(* Logix 5000 project; controller cal1615 1756-L62 rev 20.11; software revision 20.05 *)

TASK MainTask (continuous, watchdog 500 ms) : P01_System, P02_MOP_HMI_Iface, P11_Zone_1, P12_Zone_2, P13_Zone_3, P19_Advanced_Cooling, P20_Letoff, P21_Splice_Press, P22_Tension_Stand_1
TASK PIDE (periodic, rate 100 ms, priority 10, watchdog 500 ms) : P01_Main

MODULES
   Local : 1756-L62 (ICP 0, rev 20.11)
      p00_di_01 : 1756-IB16 (ICP 4, rev 3.1, Input RPI 20 ms)
           Local:4:I.DATA.0   // Digital Input Zone 1 Burner Auto
           Local:4:I.DATA.1   // Digital Input Zone 1 High Temperature Limit is Ok
           Local:4:I.DATA.2   // Digital Input Zone 1 Burner Safeties Ok
           Local:4:I.DATA.3   // Digital Input Zone 1 Recirculation Fan Rotating
           Local:4:I.DATA.4   // Digital Input Zone 1 Exhaust Fan Rotating
           Local:4:I.DATA.5   // Digital Input Zone 1 Flame Failure
           Local:4:I.DATA.6   // Digital Input Zone 1 Burner is On
           Local:4:I.DATA.7   // Digital Input Zone 1 Spare
           Local:4:I.DATA.8   // Digital Input Zone 2 Burner Auto
           Local:4:I.DATA.9   // Digital Input Zone 2 High Temperature Limit is Ok
           Local:4:I.DATA.10   // Digital Input Zone 2 Burner Safeties Ok
           Local:4:I.DATA.11   // Digital Input Zone 2 Recirculation Fan Rotating
           Local:4:I.DATA.12   // Digital Input Zone 2 Exhaust Fan Rotating
           Local:4:I.DATA.13   // Digital Input Zone 2 Flame Failure
           Local:4:I.DATA.14   // Digital Input Zone 2 Burner is On
           Local:4:I.DATA.15   // Digital Input Zone 2 Spare
      p00_di_02 : 1756-IB16 (ICP 5, rev 3.1, Input RPI 20 ms)
           Local:5:I.DATA.0   // Digital Input Zone 3 Recirculation Fan Rotating
           Local:5:I.DATA.1   // Digital Input Zone 3 Exhaust Fan Rotating
           Local:5:I.DATA.2   // Digital Input Zone 3 Spare
           Local:5:I.DATA.3   // Digital Input Zone 3 Spare
           Local:5:I.DATA.4   // Digital Input Zone 3 Spare
           Local:5:I.DATA.5   // Digital Input Zone 3 Spare
           Local:5:I.DATA.6   // Digital Input Zone 3 Spare
           Local:5:I.DATA.7   // Digital Input Zone 3 Spare
           Local:5:I.DATA.8   // Digital Input Rope Switch 1 Active
           Local:5:I.DATA.9   // Digital Input Rope Switch 2 Active
           Local:5:I.DATA.10   // Digital Input Rope Switch 3 Active
           Local:5:I.DATA.11   // Digital Input Rope Switch 4 Active
           Local:5:I.DATA.12   // Digital Input Rope Switch 5 Active
           Local:5:I.DATA.13   // Digital Input Rope Switch 6 Active
           Local:5:I.DATA.14   // Digital Input Rope Switch 7 Active
           Local:5:I.DATA.15   // Digital Input Rope Switch 8 Active
      p00_di_03 : 1756-IB16 (ICP 6, rev 3.1, Input RPI 20 ms)
           Local:6:I.DATA.0   // Digital Input Main HMI Reset PB
           Local:6:I.DATA.1   // Digital Input Main HMI Estop PB
           Local:6:I.DATA.2   // Digital Input Safety Relay 1 OK
           Local:6:I.DATA.3   // Digital Input Safety Relay 2 OK
           Local:6:I.DATA.4   // Digital Input Two Hand Safety Relay
           Local:6:I.DATA.5   // Digital Input Splice Plate High Temperature
           Local:6:I.DATA.6   // Digital Input Spare
           Local:6:I.DATA.7   // Digital Input Retraction and Rotation Fault
           Local:6:I.DATA.8   // Digital Input Spare
           Local:6:I.DATA.9   // Digital Input Spare
           Local:6:I.DATA.10   // Digital Input Spare
           Local:6:I.DATA.11   // Digital Input Spare
           Local:6:I.DATA.12   // Digital Input Spare
           Local:6:I.DATA.13   // Digital Input Spare
           Local:6:I.DATA.14   // Digital Input Spare
           Local:6:I.DATA.15   // Digital Input Spare
      p00_do_01 : 1756-OA16I (ICP 7, rev 3.1, Output RPI 20 ms)
           Local:7:O.DATA.0   // Digital Output Zone 1 Burner Enable
           Local:7:O.DATA.1   // Digital Output Zone 1 Burner Reset
           Local:7:O.DATA.2   // Digital Output Zone 2 Burner Enable
           Local:7:O.DATA.3   // Digital Output Zone 2 Burner Reset
           Local:7:O.DATA.4   // Digital Output Retraction System Motion
           Local:7:O.DATA.5   // Digital Output Spare
           Local:7:O.DATA.6   // Digital Output Spare
           Local:7:O.DATA.7   // Digital Output Spare
           Local:7:O.DATA.8   // Digital Output Spare
           Local:7:O.DATA.9   // Digital Output Spare
           Local:7:O.DATA.10   // Digital Output Spare
           Local:7:O.DATA.11   // Digital Output Spare
           Local:7:O.DATA.12   // Digital Output Spare
           Local:7:O.DATA.13   // Digital Output Spare
           Local:7:O.DATA.14   // Digital Output Spare
           Local:7:O.DATA.15   // Digital Output Spare
      Enet_A : 1756-ENBT (Ethernet 10.0.0.1, ICP 1, rev 4.1)
         p00_io_letoff : 1794-AENT (Ethernet 10.0.0.10, rev 3.1, Output RPI 25 ms)
            p00_io_letoff_di_04 : 1794-IB16 (Flex 7, rev 1.1)
                 p00_io_letoff:7:I.0   // Digital Input Impreg PB: Splice Jump
                 p00_io_letoff:7:I.1   // Digital Input Impreg SSS: Metering Rolls Open
                 p00_io_letoff:7:I.2   // Digital Input Impreg SSS: Metering Rolls Close
                 p00_io_letoff:7:I.3   // Digital Input Impreg SSS: Metering Rolls Jog FWD
                 p00_io_letoff:7:I.4   // Digital Input Impreg SSS: Metering Rolls Jog REV
                 p00_io_letoff:7:I.5   // Digital Input Impreg PP: EStop Active
                 p00_io_letoff:7:I.6   // Digital Input Impreg Spare
                 p00_io_letoff:7:I.7   // Digital Input Impreg Spare
                 p00_io_letoff:7:I.8   // Digital Input Impreg PR: Dip Tank Up
                 p00_io_letoff:7:I.9   // Digital Input Impreg PS: Enclosure Supply Filter Dirty
                 p00_io_letoff:7:I.10   // Digital Input Impreg Enclosure Supply Fan Rotating
                 p00_io_letoff:7:I.11   // Digital Input Impreg Through Tank Level Low
                 p00_io_letoff:7:I.12   // Digital Input Impreg Tank Level High
                 p00_io_letoff:7:I.13   // Digital Input Impreg Tank Level Low
                 p00_io_letoff:7:I.14   // Digital Input Impreg Spare
                 p00_io_letoff:7:I.15   // Digital Input Impreg Spare
            p00_io_letoff_do_01 : vendor 1 type 7 code 35 (Flex 3, rev 1.1)
                 p00_io_letoff:3:O.0   // Digital Output Letoff B Selected
                 p00_io_letoff:3:O.1   // Digital Output Letoff A Selected
                 p00_io_letoff:3:O.2   // Digital Output Letoff Turret in position
                 p00_io_letoff:3:O.3   // Digital Output Letoff Spare
                 p00_io_letoff:3:O.4   // Digital Output Splice Press Inlet Clamp Close
                 p00_io_letoff:3:O.5   // Digital Output Splice Press Platen Close
                 p00_io_letoff:3:O.7   // Digital Output Splice Press Exit Clamp Close
                 p00_io_letoff:3:O.8   // Digital Output Letoff Accumulator Feedroll Clutch On
                 p00_io_letoff:3:O.9   // Digital Output Letoff Accumulator Feedroll Nip Close
                 p00_io_letoff:3:O.10   // Digital Output Letoff Accumulator Tension On
                 p00_io_letoff:3:O.11   // Digital Output Letoff Accumulator Tension High/Low
                 p00_io_letoff:3:O.12   // Digital Output Tension Stand 1 Nip Close
                 p00_io_letoff:3:O.13   // Digital Output Spare
                 p00_io_letoff:3:O.14   // Digital Output Impreg Metering Rolls Close
                 p00_io_letoff:3:O.15   // Digital Output Spare
            p00_io_letoff_di_01 : 1794-IB16 (Flex 4, rev 1.1)
                 p00_io_letoff:4:I.0   // Digital Input Letoff SS: Letoff A Selected
                 p00_io_letoff:4:I.1   // Digital Input Letoff PB: Letoff A On
                 p00_io_letoff:4:I.2   // Digital Input Letoff PB: Letoff A Off Off=0
                 p00_io_letoff:4:I.3   // Digital Input Letoff PB: Letoff A Jog FWD
                 p00_io_letoff:4:I.4   // Digital Input Letoff PB: Letoff A Jog REV
                 p00_io_letoff:4:I.5   // Digital Input Letoff PB: Letoff B On
                 p00_io_letoff:4:I.6   // Digital Input Letoff PB: Letoff B Off
                 p00_io_letoff:4:I.7   // Digital Input Letoff PB: Letoff B Jog FWD
                 p00_io_letoff:4:I.8   // Digital Input Letoff PB: Letoff B Jog REV
                 p00_io_letoff:4:I.9   // Digital Input Letoff PB: Turret FWD
                 p00_io_letoff:4:I.10   // Digital Input Letoff PB: Turret REV
                 p00_io_letoff:4:I.11   // Digital Input Letoff PP: Estop Active
                 p00_io_letoff:4:I.12   // Digital Input Letoff Spare
                 p00_io_letoff:4:I.13   // Digital Input Letoff Turret in Position
                 p00_io_letoff:4:I.14   // Digital Input Letoff Spare
                 p00_io_letoff:4:I.15   // Digital Input Letoff Spare
            p00_io_letoff_di_02 : 1794-IB16 (Flex 5, rev 1.1)
                 p00_io_letoff:5:I.0   // Digital Input Splice Press Spare
                 p00_io_letoff:5:I.1   // Digital Input Splice Press Spare
                 p00_io_letoff:5:I.2   // Digital Input Splice Press PB: Open Platen
                 p00_io_letoff:5:I.3   // Digital Input Splice Press PB: Close Inlet Clamp
                 p00_io_letoff:5:I.4   // Digital Input Splice Press PB: Close Exit Clamp
                 p00_io_letoff:5:I.5   // Digital Input Splice Press PB: Feedroll Jog FWD
                 p00_io_letoff:5:I.6   // Digital Input Splice Press PB: Feedroll Jog REV
                 p00_io_letoff:5:I.7   // Digital Input Splice Press PB: Close Feedroll Nip
                 p00_io_letoff:5:I.8   // Digital Input Splice Press PB: Fill Letoff Accumulator
                 p00_io_letoff:5:I.9   // Digital Input Splice Press PP: EStop Active
                 p00_io_letoff:5:I.10   // Digital Input Splice Press Spare
                 p00_io_letoff:5:I.11   // Digital Input Accumulator Door Open
                 p00_io_letoff:5:I.12   // Digital Input Splice Press Spare
                 p00_io_letoff:5:I.13   // Digital Input Splice Press Spare
                 p00_io_letoff:5:I.14   // Digital Input Splice Press LS: Platen Closed
                 p00_io_letoff:5:I.15   // Digital Input Splice Press Spare
            p00_io_letoff_di_03 : 1794-IB16 (Flex 6, rev 1.1)
                 p00_io_letoff:6:I.0   // Digital Input Letoff Accumulator LS: Upper Limit Active
                 p00_io_letoff:6:I.1   // Digital Input Letoff Accumulator LS: Lower Limit Active
                 p00_io_letoff:6:I.2   // Digital Input Letoff Accumulator Spare
                 p00_io_letoff:6:I.3   // Digital Input Letoff Accumulator PB: Tension Stand 1 Jog FWD
                 p00_io_letoff:6:I.4   // Digital Input Letoff Accumulator PB: Tension Stand 1 Jog REV
                 p00_io_letoff:6:I.5   // Digital Input Letoff Accumulator SS: Tension Stand 1 Jog/Thread/Run Jog
                 p00_io_letoff:6:I.6   // Digital Input Letoff Accumulator SS: Tension Stand 1 Jog/Thread/Run Run
                 p00_io_letoff:6:I.7   // Digital Input Letoff Accumulator SS: Tension Stand 1 Nip Open/Auto/Close Open
                 p00_io_letoff:6:I.8   // Digital Input Letoff Accumulator SS: Tension Stand 1 Nip Open/Auto/Close Close
                 p00_io_letoff:6:I.9   // Digital Input Letoff Accumulator PP: EStop Active
                 p00_io_letoff:6:I.10   // Digital Input Letoff Accumulator Spare
                 p00_io_letoff:6:I.11   // Digital Input Letoff Accumulator Spare
                 p00_io_letoff:6:I.12   // Digital Input Letoff Accumulator Spare
                 p00_io_letoff:6:I.13   // Digital Input Letoff Accumulator Spare
                 p00_io_letoff:6:I.14   // Digital Input Letoff Accumulator Spare
                 p00_io_letoff:6:I.15   // Digital Input Letoff Accumulator Spare
            p00_io_letoff_ao_01 : 1794-OE4 (Flex 0, rev 2.1, Output RPI 80 ms)
                 p00_io_letoff:0:O.CH0DATA   // Analog Output Letoff Accumulator Counter Pressure
                 p00_io_letoff:0:O.CH1DATA   // Analog Output Letoff Accumulator Tension Pressure
                 p00_io_letoff:0:O.CH2DATA   // Analog Output Letoff Accumulator Fill Pressure
                 p00_io_letoff:0:O.CH3DATA   // Analog Output Letoff Spare
            p00_io_letoff_ai_01 : vendor 1 type 10 code 25 (Flex 1, rev 2.1, Input RPI 80 ms)
                 p00_io_letoff:1:I.CH0DATA   // Analog Input Letoff Roll Diameter
                 p00_io_letoff:1:I.CH1DATA   // Analog Input Letoff Accumulator Position
                 p00_io_letoff:1:I.CH2DATA   // Analog Input Impreg Enclosure LEL Level
                 p00_io_letoff:1:I.CH3DATA   // Analog Input Impreg Enclosure Static Pressure
                 p00_io_letoff:1:I.CH4DATA   // Analog Input Impreg Enclosure to Zone 1 Differential Pressure
                 p00_io_letoff:1:I.CH5DATA   // Analog Input Spare
                 p00_io_letoff:1:I.CH6DATA   // Analog Input Spare
                 p00_io_letoff:1:I.CH7DATA   // Analog Input Spare
            p00_io_letoff_tc_01 : vendor 1 type 10 code 28 (Flex 2, rev 1.1, Input RPI 80 ms)
                 p00_io_letoff:2:I.CH0DATA   // Thermocouple Input Splicer Platen Temperature
                 p00_io_letoff:2:I.CH1DATA   // Thermocouple Input Spare
                 p00_io_letoff:2:I.CH2DATA   // Thermocouple Input Spare
                 p00_io_letoff:2:I.CH3DATA   // Thermocouple Input Spare
                 p00_io_letoff:2:I.CH4DATA   // Thermocouple Input Spare
                 p00_io_letoff:2:I.CH5DATA   // Thermocouple Input Spare
                 p00_io_letoff:2:I.CH6DATA   // Thermocouple Input Spare
                 p00_io_letoff:2:I.CH7DATA   // Thermocouple Input Spare
                 p00_io_letoff:2:I.CH0OVERRANGEALARM   // Analog Input Splice Press TC Open Wire
                 p00_io_letoff:2:I.CH1OVERRANGEALARM   // Analog Input Spare TC Open Wire
                 p00_io_letoff:2:I.CH2OVERRANGEALARM   // Analog Input Spare TC Open Wire
                 p00_io_letoff:2:I.CH3OVERRANGEALARM   // Analog Input Spare TC Open Wire
                 p00_io_letoff:2:I.CH4OVERRANGEALARM   // Analog Input Spare TC Open Wire
                 p00_io_letoff:2:I.CH5OVERRANGEALARM   // Analog Input Spare TC Open Wire
                 p00_io_letoff:2:I.CH6OVERRANGEALARM   // Analog Input Spare TC Open Wire
                 p00_io_letoff:2:I.CH7OVERRANGEALARM   // Analog Input Spare TC Open Wire
         p00_io_oven : 1794-AENT (Ethernet 10.0.0.11, rev 3.1, Output RPI 25 ms)
            p00_io_oven_di_03 : 1794-IB16 (Flex 5, rev 1.1)
                 p00_io_oven:5:I.0   // Digital Input LS: Safety Pin 1 Stowed
                 p00_io_oven:5:I.1   // Digital Input LS: Safety Pin 2 Stowed
                 p00_io_oven:5:I.2   // Digital Input LS: Safety Pin 3 Stowed
                 p00_io_oven:5:I.3   // Digital Input LS: Safety Pin 4 Stowed
                 p00_io_oven:5:I.4   // Digital Input LS: Safety Pin 5 Stowed
                 p00_io_oven:5:I.5   // Digital Input LS: Safety Pin 6 Stowed
                 p00_io_oven:5:I.6   // Digital Input LS: Safety Pin 7 Stowed
                 p00_io_oven:5:I.7   // Digital Input LS: Safety Pin 8 Stowed
                 p00_io_oven:5:I.8   // Digital Input Spare
                 p00_io_oven:5:I.9   // Digital Input Spare
                 p00_io_oven:5:I.10   // Digital Input Spare
                 p00_io_oven:5:I.11   // Digital Input Spare
                 p00_io_oven:5:I.12   // Digital Input Spare
                 p00_io_oven:5:I.13   // Digital Input Spare
                 p00_io_oven:5:I.14   // Digital Input Spare
                 p00_io_oven:5:I.15   // Digital Input Spare
                 p00_io_oven:5:I   // Digital Input Safety Pins Stowed
            p00_io_oven_di_01 : 1794-IB16 (Flex 3, rev 1.1)
                 p00_io_oven:3:I.0   // Digital Input Zone 1 PS: Combustion Blower Pressure Ok
                 p00_io_oven:3:I.1   // Digital Input Zone 1 PS: Fresh Air Filter Dirty
                 p00_io_oven:3:I.2   // Digital Input Zone 1 PS: Combustion Blower Air Filter Dirty
                 p00_io_oven:3:I.3   // Digital Input Zone 1 PS: Recirc Fan Air Filter Dirty
                 p00_io_oven:3:I.4   // Digital Input Zone 1 LS: Access Door Open
                 p00_io_oven:3:I.5   // Digital Input Zone 1 Spare
                 p00_io_oven:3:I.6   // Digital Input Zone 1 Spare
                 p00_io_oven:3:I.7   // Digital Input Zone 1 Spare
                 p00_io_oven:3:I.8   // Digital Input Zone 2 PS: Combustion Blower Pressure Ok
                 p00_io_oven:3:I.9   // Digital Input Zone 2 PS: Filter Dirty
                 p00_io_oven:3:I.10   // Digital Input Zone 2 PS: Fresh Air Filter Dirty
                 p00_io_oven:3:I.11   // Digital Input Zone 2 PS: Recirc Fan Air Filter Dirty
                 p00_io_oven:3:I.12   // Digital Input Zone 2 LS: Access Door Open
                 p00_io_oven:3:I.13   // Digital Input Zone 2 Spare
                 p00_io_oven:3:I.14   // Digital Input Zone 2 Spare
                 p00_io_oven:3:I.15   // Digital Input Zone 2 Spare
            p00_io_oven_di_02 : 1794-IB16 (Flex 4, rev 1.1)
                 p00_io_oven:4:I.0   // Digital Input Zone 3 LS: Access Door Open
                 p00_io_oven:4:I.1   // Digital Input Zone 3 Spare
                 p00_io_oven:4:I.2   // Digital Input Zone 3 Spare
                 p00_io_oven:4:I.3   // Digital Input Retraction Control SS: Open/Off/Close Open
                 p00_io_oven:4:I.4   // Digital Input Retraction Control SS: Open/Off/Close Close
                 p00_io_oven:4:I.5   // Digital Input Retraction Control LS: Retraction Unit Up
                 p00_io_oven:4:I.6   // Digital Input Retraction Control LS: Retraction Unit Down
                 p00_io_oven:4:I.7   // Digital Input Zone 3 Filter Dirty
                 p00_io_oven:4:I.8   // Digital Input Spare
                 p00_io_oven:4:I.9   // Digital Input Spare
                 p00_io_oven:4:I.10   // Digital Input Spare
                 p00_io_oven:4:I.11   // Digital Input Spare
                 p00_io_oven:4:I.12   // Digital Input Spare
                 p00_io_oven:4:I.13   // Digital Input Spare
                 p00_io_oven:4:I.14   // Digital Input Spare
                 p00_io_oven:4:I.15   // Digital Input Spare
            p00_io_oven_ao_01 : 1794-OE4 (Flex 0, rev 2.1, Output RPI 80 ms)
                 p00_io_oven:0:O.CH0DATA   // Analog Output Zone 1 Gas Valve
                 p00_io_oven:0:O.CH1DATA   // Analog Output Zone 2 Gas Valve
                 p00_io_oven:0:O.CH2DATA   // Analog Output Zone 3 Control Valve
                 p00_io_oven:0:O.CH3DATA   // Analog Output Spare
            p00_io_oven_ai_01 : vendor 1 type 10 code 25 (Flex 1, rev 2.1, Input RPI 80 ms)
                 p00_io_oven:1:I.CH0DATA   // Analog Input Zone 1 LFL Level
                 p00_io_oven:1:I.CH1DATA   // Analog Input Zone 2 LFL Level
                 p00_io_oven:1:I.CH2DATA   // Analog Input Zone 1 to Zone 2 Differential Pressure
                 p00_io_oven:1:I.CH3DATA   // Analog Input Oxidizer Mass Flow Differential Pressure
                 p00_io_oven:1:I.CH4DATA   // Analog Input WindUp Accumulator Linear Position Transducer
                 p00_io_oven:1:I.CH5DATA   // Analog Input Spare
                 p00_io_oven:1:I.CH6DATA   // Analog Input Spare
                 p00_io_oven:1:I.CH7DATA   // Analog Input Spare
            p00_io_oven_tc_01 : vendor 1 type 10 code 28 (Flex 2, rev 1.1, Input RPI 80 ms)
                 p00_io_oven:2:I.CH0DATA   // Thermocouple Input Zone 1 Control Temperature 1
                 p00_io_oven:2:I.CH1DATA   // Thermocouple Input Zone 1 Control Temperature 2
                 p00_io_oven:2:I.CH2DATA   // Thermocouple Input Zone 2 Control Temperature 1
                 p00_io_oven:2:I.CH3DATA   // Thermocouple Input Zone 2 Control Temperature 2
                 p00_io_oven:2:I.CH4DATA   // Thermocouple Input Zone 3 Control Temperature 1
                 p00_io_oven:2:I.CH5DATA   // Thermocouple Input Zone 3 Control Temperature 2
                 p00_io_oven:2:I.CH6DATA   // Thermocouple Input Oxidizer Mass Flow Temperature
                 p00_io_oven:2:I.CH7DATA   // Thermocouple Input Spare
                 p00_io_oven:2:I.CH0OVERRANGEALARM   // Digital Input Zone 1 Control Thermocouple 1 Open Wire
                 p00_io_oven:2:I.CH1OVERRANGEALARM   // Digital Input Zone 1 Control Thermocouple 2 Open Wire
                 p00_io_oven:2:I.CH2OVERRANGEALARM   // Digital Input Zone 2 Control Thermocouple 1 Open Wire
                 p00_io_oven:2:I.CH3OVERRANGEALARM   // Digital Input Zone 2 Control Thermocouple 2 Open Wire
                 p00_io_oven:2:I.CH4OVERRANGEALARM   // Digital Input Zone 3 Control Thermocouple 1 Open Wire
                 p00_io_oven:2:I.CH5OVERRANGEALARM   // Digital Input Zone 3 Control Thermocouple 2 Open Wire
                 p00_io_oven:2:I.CH6OVERRANGEALARM   // Digital Input Zone 3 Oxidizer Mass Flow TC Open Wire
                 p00_io_oven:2:I.CH7OVERRANGEALARM   // Digital Input Zone 3 Spare TC Open Wire
         p00_io_winder : 1794-AENT (Ethernet 10.0.0.12, rev 3.1, Output RPI 25 ms)
            p00_io_winder_di_01 : 1794-IB16 (Flex 5, rev 1.1)
                 p00_io_winder:5:I.0   // Digital Input Upper poly tension A On
                 p00_io_winder:5:I.1   // Digital Input Upper poly tension B On
                 p00_io_winder:5:I.2   // Digital Input Lower poly tension A On
                 p00_io_winder:5:I.3   // Digital Input Lower poly tension B On
                 p00_io_winder:5:I.4   // Digital Input Edge Control PP: EStop Active
                 p00_io_winder:5:I.5   // Digital Input Winder Accumulator Empty
                 p00_io_winder:5:I.6   // Digital Input Windup Accumulator Off/On Selector Switch
                 p00_io_winder:5:I.7   // Digital Input Windup Accumulator Line Stop Pushbutton
                 p00_io_winder:5:I.8   // Digital Input Tension Stand 2 PB: Jog FWD
                 p00_io_winder:5:I.9   // Digital Input Tension Stand 2 PB: Jog REV
                 p00_io_winder:5:I.10   // Digital Input Tension Stand 2 SS: Jog/Thread/Run Jog
                 p00_io_winder:5:I.11   // Digital Input Tension Stand 2 SS: Jog/Thread/Run Run
                 p00_io_winder:5:I.12   // Digital Input Tension Stand 2 PP: EStop Active
                 p00_io_winder:5:I.13   // Digital Input Windup Accumulator SS: Outfeed Nip Auto
                 p00_io_winder:5:I.14   // Digital Input Windup Accumulator SS: Outfeed Nip Close
                 p00_io_winder:5:I.15   // Digital Input Windup Accumulator: OP Station E-Stop
            p00_io_winder_di_02 : 1794-IB16 (Flex 6, rev 1.1)
                 p00_io_winder:6:I.0   // Digital Input Winder Accumulator Full
                 p00_io_winder:6:I.1   // Digital Input Winder: SS: Winder A/B Winder B
                 p00_io_winder:6:I.2   // Digital Input Winder SS: Winder A Core Size Selector 3" or 6" 6" Selected
                 p00_io_winder:6:I.3   // Digital Input Winder PB: Winder A Reset Core
                 p00_io_winder:6:I.4   // Digital Input Winder PB: Winder A Jog FWD
                 p00_io_winder:6:I.5   // Digital Input Winder PB: Winder A Jog REV
                 p00_io_winder:6:I.6   // Digital Input Winder SS: Winder B Core Size Selector 3" or 6" 6" Selected
                 p00_io_winder:6:I.7   // Digital Input Winder PB: Winder B Reset Core
                 p00_io_winder:6:I.8   // Digital Input Winder PB: Winder B Jog FWD
                 p00_io_winder:6:I.9   // Digital Input Winder PB: Winder B Jog REV
                 p00_io_winder:6:I.10   // Digital Input Winder PB: Turret FWD
                 p00_io_winder:6:I.11   // Digital Input Winder PB: Turret REV
                 p00_io_winder:6:I.12   // Digital Input Winder PP: EStop Active
                 p00_io_winder:6:I.13   // Turret In Position Bit 1
                 p00_io_winder:6:I.14   // Turret In Position Bit 2
                 p00_io_winder:6:I.15   // Turret In Position Bit 3
            p00_io_winder_do_01 : vendor 1 type 7 code 35 (Flex 4, rev 1.1)
                 p00_io_winder:4:O.0   // Digital Output Spare
                 p00_io_winder:4:O.1   // Digital Output Spare
                 p00_io_winder:4:O.2   // Digital Output Winder A selected
                 p00_io_winder:4:O.3   // Digital Output Winder B selected
                 p00_io_winder:4:O.4   // Digital Output Turret in position
                 p00_io_winder:4:O.5   // Digital Output WAC Nip Close
                 p00_io_winder:4:O.6   // Digital Output WAC Nip Mode Selector Indicator Light
                 p00_io_winder:4:O.7   // Digital Output WAC Accumulator On
                 p00_io_winder:4:O.8   // Digital Output Spare
                 p00_io_winder:4:O.9   // Digital Output Spare
                 p00_io_winder:4:O.10   // Digital Output Spare
                 p00_io_winder:4:O.11   // Digital Output Spare
                 p00_io_winder:4:O.12   // Digital Output Spare
                 p00_io_winder:4:O.13   // Digital Output Spare
                 p00_io_winder:4:O.14   // Digital Output Spare
                 p00_io_winder:4:O.15   // Digital Output Spare
            p00_io_winder_ao_01 : 1794-OE4 (Flex 0, rev 2.1, Output RPI 80 ms)
                 p00_io_winder:0:O.CH0DATA   // Analog Output Upper Liner Letoff Brake A
                 p00_io_winder:0:O.CH1DATA   // Analog Output Upper Liner Letoff Brake B
                 p00_io_winder:0:O.CH2DATA   // Analog Output Lower Liner Letoff Brake A
                 p00_io_winder:0:O.CH3DATA   // Analog Output Lower Liner Letoff Brake B
            p00_io_winder_ao_02 : 1794-OE4 (Flex 1, rev 2.1, Output RPI 80 ms)
                 p00_io_winder:1:O.CH0DATA   // Analog Output Advanced Roll Cooling Pressure
                 p00_io_winder:1:O.CH1DATA   // Analog Output Advanced Roll Cooling Control Valve
                 p00_io_winder:1:O.CH2DATA   // Analog Output Windup Accumulator Tension Control I/P Converter
                 p00_io_winder:1:O.CH3DATA   // Analog Output Windup Accumulator Carriage Counter Pressure I/P Converter
            p00_io_winder_ai_01 : vendor 1 type 10 code 25 (Flex 2, rev 2.1, Input RPI 80 ms)
                 p00_io_winder:2:I.CH0DATA   // Analog Input Upper Liner Letoff A Diameter
                 p00_io_winder:2:I.CH1DATA   // Analog Input Upper Liner Letoff B Diameter
                 p00_io_winder:2:I.CH2DATA   // Analog Input Lower Liner Letoff A Diameter
                 p00_io_winder:2:I.CH3DATA   // Analog Input Lower Liner Letoff B Diameter
                 p00_io_winder:2:I.CH4DATA   // Analog Input Tension Stand 2 Load Cell
                 p00_io_winder:2:I.CH5DATA   // Analog Input Winder Roll Diameter
                 p00_io_winder:2:I.CH6DATA   // Analog Input Spare
                 p00_io_winder:2:I.CH7DATA   // Analog Input Advanced Roll Cooling Pressure
            p00_io_winder_tc_01 : vendor 1 type 10 code 28 (Flex 3, rev 1.1, Input RPI 80 ms)
                 p00_io_winder:3:I.CH0DATA   // Thermocouple Input Advanced Cooling Temperature 1
                 p00_io_winder:3:I.CH1DATA   // Thermocouple Input Advanced Cooling Temperature 2
                 p00_io_winder:3:I.CH2DATA   // Thermocouple Input Spare
                 p00_io_winder:3:I.CH3DATA   // Thermocouple Input Spare
                 p00_io_winder:3:I.CH4DATA   // Thermocouple Input Spare
                 p00_io_winder:3:I.CH5DATA   // Thermocouple Input Spare
                 p00_io_winder:3:I.CH6DATA   // Thermocouple Input Spare
                 p00_io_winder:3:I.CH7DATA   // Thermocouple Input Spare
                 p00_io_winder:3:I.CH0OVERRANGEALARM   // Digital Input Advanced Cooling Temperature 1 Open Wire
                 p00_io_winder:3:I.CH1OVERRANGEALARM   // Digital Input Advanced Cooling Temperature 2 Open Wire
                 p00_io_winder:3:I.CH2OVERRANGEALARM   // Digital Input Spare Open Wire
                 p00_io_winder:3:I.CH3OVERRANGEALARM   // Digital Input Spare Open Wire
                 p00_io_winder:3:I.CH4OVERRANGEALARM   // Digital Input Spare Open Wire
                 p00_io_winder:3:I.CH5OVERRANGEALARM   // Digital Input Spare Open Wire
                 p00_io_winder:3:I.CH6OVERRANGEALARM   // Digital Input Spare Open Wire
                 p00_io_winder:3:I.CH7OVERRANGEALARM   // Digital Input Spare Open Wire
         p00_io_line : 1794-AENT (Ethernet 10.0.0.13, rev 3.1, Output RPI 25 ms)
            p00_io_line_di_01 : 1794-IB16 (Flex 2, rev 1.1)
                 p00_io_line:2:I.0   // Digital Input Line Drive Letoff A Motor Thermostat
                 p00_io_line:2:I.1   // Digital Input Line Drive Letoff A/B Brake Thermostat
                 p00_io_line:2:I.2   // Digital Input Line Drive Letoff B Motor Thermostat
                 p00_io_line:2:I.3   // Spare
                 p00_io_line:2:I.4   // Digital Input Line Drive Letoff Turret Motor Thermostat
                 p00_io_line:2:I.5   // Digital Input Line Drive Tension Stand 1 Motor Thermostat
                 p00_io_line:2:I.6   // Digital Input Line Drive TS 1& Metering Roll Brake Thermostat
                 p00_io_line:2:I.7   // Digital Input Line Drive Metering Rolls Motor Thermostat
                 p00_io_line:2:I.8   // Spare
                 p00_io_line:2:I.9   // Digital Input Line Drive Metering Rolls Servo Operator Side Ok
                 p00_io_line:2:I.10   // Digital Input Line Drive Metering Rolls Servo Drive Side Ok
                 p00_io_line:2:I.11   // Digital Input Line Drive Tension Stand 2 Motor Thermostat
                 p00_io_line:2:I.12   // Digital Input Line Drive TS2 & Slitter Brake Thermostat
                 p00_io_line:2:I.13   // Digital Input Line Drive Slitter Motor Thermostat
                 p00_io_line:2:I.14   // Spare
                 p00_io_line:2:I.15   // Digital Input Line Drive Winder Turret Motor Thermostat
            p00_io_line_di_02 : 1794-IB16 (Flex 3, rev 1.1)
                 p00_io_line:3:I.0   // Digital Input Line Drive Winder A Motot Thermostat
                 p00_io_line:3:I.1   // Digital Input Line Drive Winder A/B Brake Thermostat
                 p00_io_line:3:I.2   // Digital Input Line Drive Winder B Motor Thermostat
                 p00_io_line:3:I.3   // Digital Input Line Drive Winder B Brake Thermostat
                 p00_io_line:3:I.4   // Digital Input Line Drive Spare
                 p00_io_line:3:I.5   // Digital Input Line Drive Spare
                 p00_io_line:3:I.6   // Digital Input Line Drive Spare
                 p00_io_line:3:I.7   // Digital Input Line Drive Spare
                 p00_io_line:3:I.8   // Digital Input Line Drive Spare
                 p00_io_line:3:I.9   // Digital Input Line Drive Spare
                 p00_io_line:3:I.10   // Digital Input Line Drive Spare
                 p00_io_line:3:I.11   // Digital Input Line Drive Spare
                 p00_io_line:3:I.12   // Digital Input Line Drive Spare
                 p00_io_line:3:I.13   // Digital Input Line Drive Spare
                 p00_io_line:3:I.14   // Digital Input Line Drive Spare
                 p00_io_line:3:I.15   // Digital Input Line Drive Spare
            p00_io_line_do_01 : vendor 1 type 7 code 35 (Flex 1, rev 1.1)
                 p00_io_line:1:O.0   // Digital Output Spare
                 p00_io_line:1:O.1   // Digital Output Line Drive Letoff Accumulator Feed Roll Reverse
                 p00_io_line:1:O.2   // Digital Output Line Drive Letoff Accumulator Feed Roll Forward
                 p00_io_line:1:O.3   // Digital Output Spare
                 p00_io_line:1:O.4   // Digital Output Spare
                 p00_io_line:1:O.5   // Digital Output Spare
                 p00_io_line:1:O.6   // Digital Output Line Drive IR Heater Enable
                 p00_io_line:1:O.7   // Digital Output Spare
                 p00_io_line:1:O.8   // Digital Output Spare
                 p00_io_line:1:O.9   // Digital Output Spare
                 p00_io_line:1:O.10   // Digital Output Spare
                 p00_io_line:1:O.11   // Digital Output Spare
                 p00_io_line:1:O.12   // Digital Output Spare
                 p00_io_line:1:O.13   // Digital Output Spare
                 p00_io_line:1:O.14   // Digital Output Spare
                 p00_io_line:1:O.15   // Digital Output Spare
            p00_io_line_ao_01 : 1794-OE4 (Flex 0, rev 2.1, Output RPI 80 ms)
                 p00_io_line:0:O.CH0DATA   // Analog Output Line Drive Splice Platen IR Heater Control
                 p00_io_line:0:O.CH1DATA   // Analog Output Line Drive Spare
                 p00_io_line:0:O.CH2DATA   // Analog Output Line Drive Spare
                 p00_io_line:0:O.CH3DATA   // Analog Output Line Drive Spare
         p00_io_prc : 1794-AENT (Ethernet 10.0.0.14, rev 3.1, Output RPI 25 ms)
            p00_io_prc_do_01 : vendor 1 type 7 code 35 (Flex 0, rev 1.1)
                 p00_io_prc:0:O.0   // Digital Output Process Drive Impreg Enclosure Exhaust Fan
                 p00_io_prc:0:O.1   // Digital Output Process Drive Spare
                 p00_io_prc:0:O.2   // Digital Output Process Drive Spare
                 p00_io_prc:0:O.3   // Digital Output Process Drive Retraction REV
                 p00_io_prc:0:O.4   // Digital Output Process Drive Retraction FWD
                 p00_io_prc:0:O.5   // Digital Output Process Drive Advanced Cooling Pump
                 p00_io_prc:0:O.6   // Digital Output Process Drive Spare
                 p00_io_prc:0:O.7   // Digital Output Process Drive Spare
                 p00_io_prc:0:O.8   // Digital Output Process Drive Spare
                 p00_io_prc:0:O.9   // Digital Output Process Drive Spare
                 p00_io_prc:0:O.10   // Digital Output Process Drive Spare
                 p00_io_prc:0:O.11   // Digital Output Process Drive Spare
                 p00_io_prc:0:O.12   // Digital Output Process Drive Spare
                 p00_io_prc:0:O.13   // Digital Output Process Drive Spare
                 p00_io_prc:0:O.14   // Digital Output Process Drive Spare
                 p00_io_prc:0:O.15   // Digital Output Process Drive Spare
            p00_io_prc_di_01 : 1794-IB16 (Flex 1, rev 1.1)
                 p00_io_prc:1:I.0   // Digital Input Process Drive Impreg Enclosure Supply Fan Motor Thermostat
                 p00_io_prc:1:I.1   // Digital Input Process Drive Zone 1 Recirc Fan Motor Thermostat
                 p00_io_prc:1:I.2   // Digital Input Process Drive Zone 1 Exhaust Fan Motor Thermostat
                 p00_io_prc:1:I.3   // Digital Input Process Drive Zone 2 Recirc Fan Motor Thermostat
                 p00_io_prc:1:I.4   // Digital Input Process Drive Zone 2 Exhaust Fan Motor Thermostat
                 p00_io_prc:1:I.5   // Digital Input Process Drive Zone 3 Recirc Fan Motor Thermostat
                 p00_io_prc:1:I.6   // Digital Input Process Drive Zone 3 Exhaust Fan Motor Thermostat
                 p00_io_prc:1:I.7   // Digital Input Process Drive Spare
                 p00_io_prc:1:I.8   // Digital Input Process Drive Spare
                 p00_io_prc:1:I.9   // Digital Input Process Drive Spare
                 p00_io_prc:1:I.10   // Digital Input Process Drive Spare
                 p00_io_prc:1:I.11   // Digital Input Process Drive Spare
                 p00_io_prc:1:I.12   // Digital Input Process Drive Spare
                 p00_io_prc:1:I.13   // Digital Input Process Drive Spare
                 p00_io_prc:1:I.14   // Digital Input Process Drive Spare
                 p00_io_prc:1:I.15   // Digital Input Process Drive Spare
         p00_vfd_imp_supply : ETHERNET-MODULE (Ethernet 10.0.0.50, rev 1.1, Output RPI 50 ms)
              p00_vfd_imp_supply:I.DATA[0]   // Input Impreg Supply Fan VFD Status Word
              p00_vfd_imp_supply:I.DATA[0].0   // Input Impreg Supply Fan VFD Faulted
              p00_vfd_imp_supply:I.DATA[0].1   // Input Impreg Supply Fan VFD Warning
              p00_vfd_imp_supply:I.DATA[0].2   // Input Impreg Supply Fan VFD Running Forward
              p00_vfd_imp_supply:I.DATA[0].3   // Input Impreg Supply Fan VFD Running Reverse
              p00_vfd_imp_supply:I.DATA[0].4   // Input Impreg Supply Fan VFD Ready
              p00_vfd_imp_supply:I.DATA[0].5   // Input Impreg Supply Fan VFD Control from Net
              p00_vfd_imp_supply:I.DATA[0].6   // Input Impreg Supply Fan VFD Reference from Net
              p00_vfd_imp_supply:I.DATA[0].7   // Input Impreg Supply Fan VFD At Reference
              p00_vfd_imp_supply:I.DATA[1]   // Input Impreg Supply Fan VFD Speed
              p00_vfd_imp_supply:I.DATA[2]   // Input Impreg Supply Fan VFD Amps
              p00_vfd_imp_supply:I.DATA[3]   // Input Impreg Supply Fan VFD Max Hertz
              p00_vfd_imp_supply:I.DATA[4]   // Input Impreg Supply Fan VFD Motor Nameplate Hertz
              p00_vfd_imp_supply:I.DATA[5]   // Input Impreg Supply Fan VFD Motor Nameplate RPM
              p00_vfd_imp_supply:I   // Impreg Supply Fan VFD
              p00_vfd_imp_supply:O.DATA[0]   // Output Impreg Supply Fan VFD Control Word
              p00_vfd_imp_supply:O.DATA[0].0   // Output Impreg Supply Fan VFD Run Forward
              p00_vfd_imp_supply:O.DATA[0].1   // Output Impreg Supply Fan VFD Run Reverse
              p00_vfd_imp_supply:O.DATA[0].2   // Output Impreg Supply Fan VFD Fault Reset
              p00_vfd_imp_supply:O.DATA[0].5   // Output Impreg Supply Fan VFD Net Control
              p00_vfd_imp_supply:O.DATA[0].6   // Output Impreg Supply Fan VFD Net Reference
              p00_vfd_imp_supply:O.DATA[1]   // Output Impreg Supply Fan VFD Speed Command
              p00_vfd_imp_supply:O   // Impreg Supply Fan VFD
              p00_vfd_imp_supply:C   // Tension Stand 1 VFD
         p00_vfd_z1_recirc : ETHERNET-MODULE (Ethernet 10.0.0.51, rev 1.1, Output RPI 50 ms)
              p00_vfd_z1_recirc:I.DATA[0]   // Input Zone 1 Recirc VFD Status Word
              p00_vfd_z1_recirc:I.DATA[0].0   // Input Zone 1 Recirc VFD Faulted
              p00_vfd_z1_recirc:I.DATA[0].1   // Input Zone 1 Recirc VFD Warning
              p00_vfd_z1_recirc:I.DATA[0].2   // Input Zone 1 Recirc VFD Running Forward
              p00_vfd_z1_recirc:I.DATA[0].3   // Input Zone 1 Recirc VFD Running Reverse
              p00_vfd_z1_recirc:I.DATA[0].4   // Input Zone 1 Recirc VFD Ready
              p00_vfd_z1_recirc:I.DATA[0].5   // Input Zone 1 Recirc VFD Control from Net
              p00_vfd_z1_recirc:I.DATA[0].6   // Input Zone 1 Recirc VFD Reference from Net
              p00_vfd_z1_recirc:I.DATA[0].7   // Input Zone 1 Recirc VFD At Reference
              p00_vfd_z1_recirc:I.DATA[1]   // Input Zone 1 Recirc VFD Status VFD Speed
              p00_vfd_z1_recirc:I.DATA[2]   // Input Zone 1 Recirc VFD Status VFD Amps
              p00_vfd_z1_recirc:I.DATA[3]   // Input Zone 1 Recirc VFD Status VFD Max Hertz
              p00_vfd_z1_recirc:I.DATA[4]   // Input Zone 1 Recirc VFD Status VFD Motor Nameplate Hertz
              p00_vfd_z1_recirc:I.DATA[5]   // Input Zone 1 Recirc VFD Status VFD Motor Nameplate RPM
              p00_vfd_z1_recirc:I   // Zone 1 Recirc VFD
              p00_vfd_z1_recirc:O.DATA[0]   // Output Zone 1 Recirc VFD Status VFD Control Word
              p00_vfd_z1_recirc:O.DATA[0].0   // Output Zone 1 Recirc VFD Status VFD Run Forward
              p00_vfd_z1_recirc:O.DATA[0].1   // Output Zone 1 Recirc VFD Status VFD Run Reverse
              p00_vfd_z1_recirc:O.DATA[0].2   // Output Zone 1 Recirc VFD Status VFD Fault Reset
              p00_vfd_z1_recirc:O.DATA[0].5   // Output Zone 1 Recirc VFD Status VFD Net Control
              p00_vfd_z1_recirc:O.DATA[0].6   // Output Zone 1 Recirc VFD Status VFD Net Reference
              p00_vfd_z1_recirc:O.DATA[1]   // Output Zone 1 Recirc VFD Status VFD Speed Command
              p00_vfd_z1_recirc:O   // Zone 1 Recirc VFD
              p00_vfd_z1_recirc:C   // Zone 1 Recirc VFD
         p00_vfd_z1_exhaust : ETHERNET-MODULE (Ethernet 10.0.0.52, rev 1.1, Output RPI 50 ms)
              p00_vfd_z1_exhaust:I.DATA[0]   // Input Zone 1 Exhaust VFD Status Word
              p00_vfd_z1_exhaust:I.DATA[0].0   // Input Zone 1 Exhaust VFD Faulted
              p00_vfd_z1_exhaust:I.DATA[0].1   // Input Zone 1 Exhaust VFD Warning
              p00_vfd_z1_exhaust:I.DATA[0].2   // Input Zone 1 Exhaust VFD Running Forward
              p00_vfd_z1_exhaust:I.DATA[0].3   // Input Zone 1 Exhaust VFD Running Reverse
              p00_vfd_z1_exhaust:I.DATA[0].4   // Input Zone 1 Exhaust VFD Ready
              p00_vfd_z1_exhaust:I.DATA[0].5   // Input Zone 1 Exhaust VFD Control from Net
              p00_vfd_z1_exhaust:I.DATA[0].6   // Input Zone 1 Exhaust VFD Reference from Net
              p00_vfd_z1_exhaust:I.DATA[0].7   // Input Zone 1 Exhaust VFD At Reference
              p00_vfd_z1_exhaust:I.DATA[1]   // Input Zone 1 Exhaust VFD Speed
              p00_vfd_z1_exhaust:I.DATA[2]   // Input Zone 1 Exhaust VFD Amps
              p00_vfd_z1_exhaust:I.DATA[3]   // Input Zone 1 Exhaust VFD Max Hertz
              p00_vfd_z1_exhaust:I.DATA[4]   // Input Zone 1 Exhaust VFD Motor Nameplate Hertz
              p00_vfd_z1_exhaust:I.DATA[5]   // Input Zone 1 Exhaust VFD Motor Nameplate RPM
              p00_vfd_z1_exhaust:I   // Zone 1 Exhaust VFD
              p00_vfd_z1_exhaust:O.DATA[0]   // Output Zone 1 Exhaust VFD Control Word
              p00_vfd_z1_exhaust:O.DATA[0].0   // Output Zone 1 Exhaust VFD Run Forward
              p00_vfd_z1_exhaust:O.DATA[0].1   // Output Zone 1 Exhaust VFD Run Reverse
              p00_vfd_z1_exhaust:O.DATA[0].2   // Output Zone 1 Exhaust VFD Fault Reset
              p00_vfd_z1_exhaust:O.DATA[0].5   // Output Zone 1 Exhaust VFD Net Control
              p00_vfd_z1_exhaust:O.DATA[0].6   // Output Zone 1 Exhaust VFD Net Reference
              p00_vfd_z1_exhaust:O.DATA[1]   // Output Zone 1 Exhaust VFD Speed Command
              p00_vfd_z1_exhaust:O   // Zone 1 Exhaust VFD
              p00_vfd_z1_exhaust:C   // Zone 1 Exhaust VFD
         p00_vfd_z2_recirc : ETHERNET-MODULE (Ethernet 10.0.0.53, rev 1.1, Output RPI 50 ms)
              p00_vfd_z2_recirc:I.DATA[0]   // Input Zone 2 Recirc VFD Status Word
              p00_vfd_z2_recirc:I.DATA[0].0   // Input Zone 2 Recirc VFD Faulted
              p00_vfd_z2_recirc:I.DATA[0].1   // Input Zone 2 Recirc VFD Warning
              p00_vfd_z2_recirc:I.DATA[0].2   // Input Zone 2 Recirc VFD Running Forward
              p00_vfd_z2_recirc:I.DATA[0].3   // Input Zone 2 Recirc VFD Running Reverse
              p00_vfd_z2_recirc:I.DATA[0].4   // Input Zone 2 Recirc VFD Ready
              p00_vfd_z2_recirc:I.DATA[0].5   // Input Zone 2 Recirc VFD Control from Net
              p00_vfd_z2_recirc:I.DATA[0].6   // Input Zone 2 Recirc VFD Reference from Net
              p00_vfd_z2_recirc:I.DATA[0].7   // Input Zone 2 Recirc VFD At Reference
              p00_vfd_z2_recirc:I.DATA[1]   // Input Zone 2 Recirc VFD Speed
              p00_vfd_z2_recirc:I.DATA[2]   // Input Zone 2 Recirc VFD Amps
              p00_vfd_z2_recirc:I.DATA[3]   // Input Zone 2 Recirc VFD Max Hertz
              p00_vfd_z2_recirc:I.DATA[4]   // Input Zone 2 Recirc VFD Motor Nameplate Hertz
              p00_vfd_z2_recirc:I.DATA[5]   // Input Zone 2 Recirc VFD Motor Nameplate RPM
              p00_vfd_z2_recirc:I   // Zone 2 Recirc VFD
              p00_vfd_z2_recirc:O.DATA[0]   // Output Zone 2 Recirc VFD Control Word
              p00_vfd_z2_recirc:O.DATA[0].0   // Output Zone 2 Recirc VFD Run Forward
              p00_vfd_z2_recirc:O.DATA[0].1   // Output Zone 2 Recirc VFD Run Reverse
              p00_vfd_z2_recirc:O.DATA[0].2   // Output Zone 2 Recirc VFD Fault Reset
              p00_vfd_z2_recirc:O.DATA[0].3   // Input Zone 2 Recirc VFD Running Reverse
              p00_vfd_z2_recirc:O.DATA[0].4   // Input Zone 2 Recirc VFD Ready
              p00_vfd_z2_recirc:O.DATA[0].5   // Output Zone 2 Recirc VFD Net Control
              p00_vfd_z2_recirc:O.DATA[0].6   // Output Zone 2 Recirc VFD Net Reference
              p00_vfd_z2_recirc:O.DATA[0].7   // Input Zone 2 Recirc VFD At Reference
              p00_vfd_z2_recirc:O.DATA[1]   // Output Zone 2 Recirc VFD Speed Command
              p00_vfd_z2_recirc:O.DATA[2]   // Input Zone 2 Recirc VFD Amps
              p00_vfd_z2_recirc:O.DATA[3]   // Input Zone 2 Recirc VFD Max Hertz
              p00_vfd_z2_recirc:O.DATA[4]   // Input Zone 2 Recirc VFD Motor Nameplate Hertz
              p00_vfd_z2_recirc:O.DATA[5]   // Input Zone 2 Recirc VFD Motor Nameplate RPM
              p00_vfd_z2_recirc:O   // Zone 2 Recirc VFD
              p00_vfd_z2_recirc:C   // Zone 2 Recirc VFD
         p00_vfd_z2_exhaust : ETHERNET-MODULE (Ethernet 10.0.0.54, rev 1.1, Output RPI 50 ms)
              p00_vfd_z2_exhaust:I.DATA[0]   // Input Zone 2 Exhaust VFD Status Word
              p00_vfd_z2_exhaust:I.DATA[0].0   // Input Zone 2 Exhaust VFD Faulted
              p00_vfd_z2_exhaust:I.DATA[0].1   // Input Zone 2 Exhaust VFD Warning
              p00_vfd_z2_exhaust:I.DATA[0].2   // Input Zone 2 Exhaust VFD Running Forward
              p00_vfd_z2_exhaust:I.DATA[0].3   // Input Zone 2 Exhaust VFD Running Reverse
              p00_vfd_z2_exhaust:I.DATA[0].4   // Input Zone 2 Exhaust VFD Ready
              p00_vfd_z2_exhaust:I.DATA[0].5   // Input Zone 2 Exhaust VFD Control from Net
              p00_vfd_z2_exhaust:I.DATA[0].6   // Input Zone 2 Exhaust VFD Reference from Net
              p00_vfd_z2_exhaust:I.DATA[0].7   // Input Zone 2 Exhaust VFD At Reference
              p00_vfd_z2_exhaust:I.DATA[1]   // Input Zone 2 Exhaust VFD Speed
              p00_vfd_z2_exhaust:I.DATA[2]   // Input Zone 2 Exhaust VFD Amps
              p00_vfd_z2_exhaust:I.DATA[3]   // Input Zone 2 Exhaust VFD Max Hertz
              p00_vfd_z2_exhaust:I.DATA[4]   // Input Zone 2 Exhaust VFD Motor Nameplate Hertz
              p00_vfd_z2_exhaust:I.DATA[5]   // Input Zone 2 Exhaust VFD Motor Nameplate RPM
              p00_vfd_z2_exhaust:I   // Zone 2 Exhaust VFD
              p00_vfd_z2_exhaust:O.DATA[0]   // Output Zone 2 Exhaust VFD Control Word
              p00_vfd_z2_exhaust:O.DATA[0].0   // Output Zone 2 Exhaust VFD Run Forward
              p00_vfd_z2_exhaust:O.DATA[0].1   // Output Zone 2 Exhaust VFD Run Reverse
              p00_vfd_z2_exhaust:O.DATA[0].2   // Output Zone 2 Exhaust VFD Fault Reset
              p00_vfd_z2_exhaust:O.DATA[0].5   // Output Zone 2 Exhaust VFD Net Control
              p00_vfd_z2_exhaust:O.DATA[0].6   // Output Zone 2 Exhaust VFD Net Reference
              p00_vfd_z2_exhaust:O.DATA[1]   // Output Zone 2 Exhaust VFD Speed Command
              p00_vfd_z2_exhaust:O   // Zone 2 Exhaust VFD
              p00_vfd_z2_exhaust:C   // Zone 2 Exhaust VFD
         p00_vfd_z3_recirc : ETHERNET-MODULE (Ethernet 10.0.0.55, rev 1.1, Output RPI 50 ms)
              p00_vfd_z3_recirc:I.DATA[0]   // Input Zone 3 Recirc VFD Status Word
              p00_vfd_z3_recirc:I.DATA[0].0   // Input Zone 3 Recirc VFD Faulted
              p00_vfd_z3_recirc:I.DATA[0].1   // Input Zone 3 Recirc VFD Warning
              p00_vfd_z3_recirc:I.DATA[0].2   // Input Zone 3 Recirc VFD Running Forward
              p00_vfd_z3_recirc:I.DATA[0].3   // Input Zone 3 Recirc VFD Running Reverse
              p00_vfd_z3_recirc:I.DATA[0].4   // Input Zone 3 Recirc VFD Ready
              p00_vfd_z3_recirc:I.DATA[0].5   // Input Zone 3 Recirc VFD Control from Net
              p00_vfd_z3_recirc:I.DATA[0].6   // Input Zone 3 Recirc VFD Reference from Net
              p00_vfd_z3_recirc:I.DATA[0].7   // Input Zone 3 Recirc VFD At Reference
              p00_vfd_z3_recirc:I.DATA[1]   // Input Zone 3 Recirc VFD Speed
              p00_vfd_z3_recirc:I.DATA[2]   // Input Zone 3 Recirc VFD Amps
              p00_vfd_z3_recirc:I.DATA[3]   // Input Zone 3 Recirc VFD Max Hertz
              p00_vfd_z3_recirc:I.DATA[4]   // Input Zone 3 Recirc VFD Motor Nameplate Hertz
              p00_vfd_z3_recirc:I.DATA[5]   // Input Zone 3 Recirc VFD Motor Nameplate RPM
              p00_vfd_z3_recirc:I   // Zone 3 Recirc VFD
              p00_vfd_z3_recirc:O.DATA[0]   // Output Zone 3 Recirc VFD Control Word
              p00_vfd_z3_recirc:O.DATA[0].0   // Output Zone 3 Recirc VFD Run Forward
              p00_vfd_z3_recirc:O.DATA[0].1   // Output Zone 3 Recirc VFD Run Reverse
              p00_vfd_z3_recirc:O.DATA[0].2   // Output Zone 3 Recirc VFD Fault Reset
              p00_vfd_z3_recirc:O.DATA[0].5   // Output Zone 3 Recirc VFD Net Control
              p00_vfd_z3_recirc:O.DATA[0].6   // Output Zone 3 Recirc VFD Net Reference
              p00_vfd_z3_recirc:O.DATA[1]   // Output Zone 3 Recirc VFD Speed Command
              p00_vfd_z3_recirc:O   // Zone 3 Recirc VFD
              p00_vfd_z3_recirc:C   // Zone 3 Recirc VFD
         p00_vfd_z3_exhaust : ETHERNET-MODULE (Ethernet 10.0.0.56, rev 1.1, Output RPI 50 ms)
              p00_vfd_z3_exhaust:I.DATA[0]   // Input Zone 3 Exhaust VFD Status Word
              p00_vfd_z3_exhaust:I.DATA[0].0   // Input Zone 3 Exhaust VFD Faulted
              p00_vfd_z3_exhaust:I.DATA[0].1   // Input Zone 3 Exhaust VFD Warning
              p00_vfd_z3_exhaust:I.DATA[0].2   // Input Zone 3 Exhaust VFD Running Forward
              p00_vfd_z3_exhaust:I.DATA[0].3   // Input Zone 3 Exhaust VFD Running Reverse
              p00_vfd_z3_exhaust:I.DATA[0].4   // Input Zone 3 Exhaust VFD Ready
              p00_vfd_z3_exhaust:I.DATA[0].5   // Input Zone 3 Exhaust VFD Control from Net
              p00_vfd_z3_exhaust:I.DATA[0].6   // Input Zone 3 Exhaust VFD Reference from Net
              p00_vfd_z3_exhaust:I.DATA[0].7   // Input Zone 3 Exhaust VFD At Reference
              p00_vfd_z3_exhaust:I.DATA[1]   // Input Zone 3 Exhaust VFD Speed
              p00_vfd_z3_exhaust:I.DATA[2]   // Input Zone 3 Exhaust VFD Amps
              p00_vfd_z3_exhaust:I.DATA[3]   // Input Zone 3 Exhaust VFD Max Hertz
              p00_vfd_z3_exhaust:I.DATA[4]   // Input Zone 3 Exhaust VFD Motor Nameplate Hertz
              p00_vfd_z3_exhaust:I.DATA[5]   // Input Zone 3 Exhaust VFD Motor Nameplate RPM
              p00_vfd_z3_exhaust:I   // Zone 3 Exhaust VFD
              p00_vfd_z3_exhaust:O.DATA[0]   // Output Zone 3 Exhaust VFD Control Word
              p00_vfd_z3_exhaust:O.DATA[0].0   // Output Zone 3 Exhaust VFD Run Forward
              p00_vfd_z3_exhaust:O.DATA[0].1   // Output Zone 3 Exhaust VFD Run Reverse
              p00_vfd_z3_exhaust:O.DATA[0].2   // Output Zone 3 Exhaust VFD Fault Reset
              p00_vfd_z3_exhaust:O.DATA[0].5   // Output Zone 3 Exhaust VFD Net Control
              p00_vfd_z3_exhaust:O.DATA[0].6   // Output Zone 3 Exhaust VFD Net Reference
              p00_vfd_z3_exhaust:O.DATA[1]   // Output Zone 3 Exhaust VFD Speed Command
              p00_vfd_z3_exhaust:O   // Zone 3 Exhaust VFD
              p00_vfd_z3_exhaust:C   // Zone 3 Exhaust VFD
         p00_vfd_wdb : ETHERNET-MODULE (Ethernet 10.0.0.60, rev 1.1, Output RPI 10 ms)
              p00_vfd_wdb:I.DATA[0]   // Input Winder B VFD Status Word
              p00_vfd_wdb:I.DATA[0].0   // Input Winder B VFD Faulted
              p00_vfd_wdb:I.DATA[0].1   // Input Winder B VFD Warning
              p00_vfd_wdb:I.DATA[0].2   // Input Winder B VFD Running Forward
              p00_vfd_wdb:I.DATA[0].3   // Input Winder B VFD Running Reverse
              p00_vfd_wdb:I.DATA[0].4   // Input Winder B VFD Ready
              p00_vfd_wdb:I.DATA[0].5   // Input Winder B VFD Control from Net
              p00_vfd_wdb:I.DATA[0].6   // Input Winder B VFD Reference from Net
              p00_vfd_wdb:I.DATA[0].7   // Input Winder B VFD At Reference
              p00_vfd_wdb:I.DATA[1]   // Input Winder B VFD Speed
              p00_vfd_wdb:I.DATA[2]   // Input Winder B VFD Amps
              p00_vfd_wdb:I.DATA[3]   // Input Winder B VFD Max Hertz
              p00_vfd_wdb:I.DATA[4]   // Input Winder B VFD Motor Nameplate Hertz
              p00_vfd_wdb:I.DATA[5]   // Input Winder B VFD Motor Nameplate RPM
              p00_vfd_wdb:I   // Winder B VFD
              p00_vfd_wdb:O.DATA[0]   // Output Winder B VFD Control Word
              p00_vfd_wdb:O.DATA[0].0   // Output Winder B VFD Run Forward
              p00_vfd_wdb:O.DATA[0].1   // Output Winder B VFD Run Reverse
              p00_vfd_wdb:O.DATA[0].2   // Output Winder B VFD Fault Reset
              p00_vfd_wdb:O.DATA[0].5   // Output Winder B VFD Net Control
              p00_vfd_wdb:O.DATA[0].6   // Output Winder B VFD Net Reference
              p00_vfd_wdb:O.DATA[1]   // Output Winder B VFD Speed Command
              p00_vfd_wdb:O   // Winder B VFD
              p00_vfd_wdb:C   // Winder B VFD
      Enet_B : 1756-ENBT (ICP 2, Ethernet 10.0.1.1, rev 4.1)
         p00_vfd_loa : ETHERNET-MODULE (Ethernet 10.0.1.10, rev 1.1, Output RPI 10 ms)
              p00_vfd_loa:I   // Winder Winder B Speed Control Speed Offset
              p00_vfd_loa:C   // Letoff A VFD
         p00_vfd_lob : ETHERNET-MODULE (Ethernet 10.0.1.11, rev 1.1, Output RPI 10 ms)
              p00_vfd_lob:I.DATA[0]   // Input Letoff B VFD Status Word
              p00_vfd_lob:I.DATA[0].0   // Input Letoff B VFD Faulted
              p00_vfd_lob:I.DATA[0].1   // Input Letoff B VFD Warning
              p00_vfd_lob:I.DATA[0].2   // Input Letoff B VFD Running Forward
              p00_vfd_lob:I.DATA[0].3   // Input Letoff B VFD Running Reverse
              p00_vfd_lob:I.DATA[0].4   // Input Letoff B VFD Ready
              p00_vfd_lob:I.DATA[0].5   // Input Letoff B VFD Control from Net
              p00_vfd_lob:I.DATA[0].6   // Input Letoff B VFD Reference from Net
              p00_vfd_lob:I.DATA[0].7   // Input Letoff B VFD At Reference
              p00_vfd_lob:I.DATA[1]   // Input Letoff B VFD Speed
              p00_vfd_lob:I.DATA[2]   // Input Letoff B VFD Amps
              p00_vfd_lob:I.DATA[3]   // Input Letoff B VFD Max Hertz
              p00_vfd_lob:I.DATA[4]   // Input Letoff B VFD Motor Nameplate Hertz
              p00_vfd_lob:I.DATA[5]   // Input Letoff B VFD Motor Nameplate RPM
              p00_vfd_lob:I   // Letoff B VFD
              p00_vfd_lob:O.DATA[0]   // Output Tension Stand 1 VFD Control Word
              p00_vfd_lob:O.DATA[0].0   // Output Letoff B VFD Run Forward
              p00_vfd_lob:O.DATA[0].1   // Output Letoff B VFD Run Reverse
              p00_vfd_lob:O.DATA[0].2   // Output Letoff B VFD Fault Reset
              p00_vfd_lob:O.DATA[0].5   // Output Letoff B VFD Net Control
              p00_vfd_lob:O.DATA[0].6   // Output Letoff B VFD Net Reference
              p00_vfd_lob:O.DATA[1]   // Output Letoff B VFD Speed Command
              p00_vfd_lob:O   // Letoff B VFD
              p00_vfd_lob:C   // Letoff B VFD
         p00_vfd_lo_turret : ETHERNET-MODULE (Ethernet 10.0.1.12, rev 1.1, Output RPI 10 ms)
              p00_vfd_lo_turret:I.DATA[0]   // Input Letoff Turret VFD Status Word
              p00_vfd_lo_turret:I.DATA[0].0   // Input Letoff Turret VFD Faulted
              p00_vfd_lo_turret:I.DATA[0].1   // Input Letoff Turret VFD Warning
              p00_vfd_lo_turret:I.DATA[0].2   // Input Letoff Turret VFD Running Forward
              p00_vfd_lo_turret:I.DATA[0].3   // Input Letoff Turret VFD Running Reverse
              p00_vfd_lo_turret:I.DATA[0].4   // Input Letoff Turret VFD Ready
              p00_vfd_lo_turret:I.DATA[0].5   // Input Letoff Turret VFD Control from Net
              p00_vfd_lo_turret:I.DATA[0].6   // Input Letoff Turret VFD Reference from Net
              p00_vfd_lo_turret:I.DATA[0].7   // Input Letoff Turret VFD At Reference
              p00_vfd_lo_turret:I.DATA[1]   // Input Letoff Turret VFD Speed
              p00_vfd_lo_turret:I.DATA[2]   // Input Letoff Turret VFD Amps
              p00_vfd_lo_turret:I.DATA[3]   // Input Letoff Turret VFD Max Hertz
              p00_vfd_lo_turret:I.DATA[4]   // Input Letoff Turret VFD Motor Nameplate Hertz
              p00_vfd_lo_turret:I.DATA[5]   // Input Letoff Turret VFD Motor Nameplate RPM
              p00_vfd_lo_turret:I   // Letoff Turret VFD
              p00_vfd_lo_turret:O.DATA[0]   // Output Letoff Turret VFD Control Word
              p00_vfd_lo_turret:O.DATA[0].0   // Output Letoff Turret VFD Run Forward
              p00_vfd_lo_turret:O.DATA[0].1   // Output Letoff Turret VFD Run Reverse
              p00_vfd_lo_turret:O.DATA[0].2   // Output Letoff Turret VFD Fault Reset
              p00_vfd_lo_turret:O.DATA[0].5   // Output Letoff Turret VFD Net Control
              p00_vfd_lo_turret:O.DATA[0].6   // Output Letoff Turret VFD Net Reference
              p00_vfd_lo_turret:O.DATA[1]   // Output Letoff Turret VFD Speed Command
              p00_vfd_lo_turret:O   // Letoff Turret VFD
              p00_vfd_lo_turret:C   // Letoff Turret VFD
         p00_vfd_ts1 : ETHERNET-MODULE (Ethernet 10.0.1.13, rev 1.1, Output RPI 10 ms)
              p00_vfd_ts1:C   // Tension Stand 1 VFD
         p00_vfd_mtr : ETHERNET-MODULE (Ethernet 10.0.1.14, rev 1.1, Output RPI 10 ms)
              p00_vfd_mtr:I.DATA[0]   // Input Impreg Metering VFD Status Word
              p00_vfd_mtr:I.DATA[0].0   // Input Impreg Metering VFD Faulted
              p00_vfd_mtr:I.DATA[0].1   // Input Impreg Metering VFD Warning
              p00_vfd_mtr:I.DATA[0].2   // Input Impreg Metering VFD Running Forward
              p00_vfd_mtr:I.DATA[0].3   // Input Impreg Metering VFD Running Reverse
              p00_vfd_mtr:I.DATA[0].4   // Input Impreg Metering VFD Ready
              p00_vfd_mtr:I.DATA[0].5   // Input Impreg Metering VFD Control from Net
              p00_vfd_mtr:I.DATA[0].6   // Input Impreg Metering VFD Reference from Net
              p00_vfd_mtr:I.DATA[0].7   // Input Impreg Metering VFD At Reference
              p00_vfd_mtr:I.DATA[1]   // Input Impreg Metering VFD Speed
              p00_vfd_mtr:I.DATA[2]   // Input Impreg Metering VFD Amps
              p00_vfd_mtr:I.DATA[3]   // Input Impreg Metering VFD Max Hertz
              p00_vfd_mtr:I.DATA[4]   // Input Impreg Metering VFD Motor Nameplate Hertz
              p00_vfd_mtr:I.DATA[5]   // Input Impreg Metering VFD Motor Nameplate RPM
              p00_vfd_mtr:I   // Metering Roll VFD
              p00_vfd_mtr:O.DATA[0]   // Output Impreg Metering VFDControl Word
              p00_vfd_mtr:O.DATA[0].0   // Output Impreg Metering VFD Run Forward
              p00_vfd_mtr:O.DATA[0].1   // Output Impreg Metering VFD Run Reverse
              p00_vfd_mtr:O.DATA[0].2   // Output Impreg Metering VFD Fault Reset
              p00_vfd_mtr:O.DATA[0].5   // Output Impreg Metering VFD Net Control
              p00_vfd_mtr:O.DATA[0].6   // Output Impreg Metering VFD Net Reference
              p00_vfd_mtr:O.DATA[1]   // Output Impreg Metering VFD Speed Command
              p00_vfd_mtr:O   // Output Impreg Metering VFD
              p00_vfd_mtr:C   // Metering Roll VFD
         p00_srv_mtr_os : ETHERNET-MODULE (Ethernet 10.0.1.15, rev 1.1, Output RPI 10 ms)
              p00_srv_mtr_os:I.DATA[0]   // Input Mayer Rod Operator Status Word
              p00_srv_mtr_os:I.DATA[0].0   // Input Mayer Rod Operator Side Operation Mode Bit 0
              p00_srv_mtr_os:I.DATA[0].1   // Input Mayer Rod Operator Side Operation Mode Bit 1
              p00_srv_mtr_os:I.DATA[0].2   // Input Mayer Rod Operator Side Homed
              p00_srv_mtr_os:I.DATA[0].3   // Input Mayer Rod Operator Side Stand Still
              p00_srv_mtr_os:I.DATA[0].4   // Input Mayer Rod Operator Side Target Position Reached
              p00_srv_mtr_os:I.DATA[0].5   // Input Mayer Rod Operator Side Command Change Bit
              p00_srv_mtr_os:I.DATA[0].6   // Input Mayer Rod Operator Side Operating Mode Error
              p00_srv_mtr_os:I.DATA[0].7   // Input Mayer Rod Operator Side Drive does not follow command value (e.g. when Drive Halt is active)
              p00_srv_mtr_os:I.DATA[0].8   // Input Mayer Rod Operator Side Actual Operating Mode
              p00_srv_mtr_os:I.DATA[0].9   // Input Mayer Rod Operator Side Actual Operating Mode
              p00_srv_mtr_os:I.DATA[0].10   // Input Mayer Rod Operator Side
              p00_srv_mtr_os:I.DATA[0].11   // Input Mayer Rod Operator Side Class 3 Diagnostic Message
              p00_srv_mtr_os:I.DATA[0].12   // Input Mayer Rod Operator Side Class 2 Diagnostic Message
              p00_srv_mtr_os:I.DATA[0].13   // Input Mayer Rod Operator Side Class 1 Diagnostic Message
              p00_srv_mtr_os:I.DATA[0].14   // Input Mayer Rod Operator Side Ready for Operation Bit 14/15 00: Not Ready 01:(bb) 10: (Ab) 11: (AF)
              p00_srv_mtr_os:I.DATA[0].15   // Input Mayer Rod Operator Side Ready for Operation Bit 14/15 00: Not Ready 01:(bb) 10: (Ab) 11: (AF)
              p00_srv_mtr_os:I.DATA[1]   // Input Mayer Rod Operator Side Velocity Feedback
              p00_srv_mtr_os:I.DATA[2]   // Input Mayer Rod Operator Side Position Feedback
              p00_srv_mtr_os:I.DATA[3]   // Input Mayer Rod Operator Side Torque Feedback
              p00_srv_mtr_os:I.DATA[4]   // Input Mayer Rod Operator Side Error Message
              p00_srv_mtr_os:I.DATA[4].1   // Input Mayer Rod Operator Side Amplifier Overtemperature Shutdown
              p00_srv_mtr_os:I.DATA[4].2   // Input Mayer Rod Operator Side Motot Overtemperature Shutdown
              p00_srv_mtr_os:I.DATA[4].3   // Input Mayer Rod Operator Side Reserved
              p00_srv_mtr_os:I.DATA[4].4   // Input Mayer Rod Operator Side Control Voltage Error
              p00_srv_mtr_os:I.DATA[4].5   // Input Mayer Rod Operator Side Encoder Error
              p00_srv_mtr_os:I.DATA[4].6   // Input Mayer Rod Operator Side Reserved
              p00_srv_mtr_os:I.DATA[4].7   // Input Mayer Rod Operator Side Overcurrent Error
              p00_srv_mtr_os:I.DATA[4].8   // Input Mayer Rod Operator Side Reserved
              p00_srv_mtr_os:I.DATA[4].9   // Input Mayer Rod Operator Side Undervoltage Error
              p00_srv_mtr_os:I.DATA[4].10   // Input Mayer Rod Operator Side Reserved
              p00_srv_mtr_os:I.DATA[4].11   // Input Mayer Rod Operator Side Excessive Deviation
              p00_srv_mtr_os:I.DATA[4].12   // Input Mayer Rod Operator Side Communication Error
              p00_srv_mtr_os:I.DATA[4].13   // Input Mayer Rod Operator Side Position Limit Value Exceeded
              p00_srv_mtr_os:I.DATA[4].14   // Input Mayer Rod Operator Side Reserved
              p00_srv_mtr_os:I.DATA[4].15   // Input Mayer Rod Operator Side Manufacturer- Specific Error
              p00_srv_mtr_os:I.DATA[5]   // Input Mayer Rod Operator Side Warning Message
              p00_srv_mtr_os:I.DATA[5].0   // Input Mayer Rod Operator Side Overload Warning
              p00_srv_mtr_os:I.DATA[5].1   // Input Mayer Rod Operator Side Amplifier Overtemperature Warning
              p00_srv_mtr_os:I.DATA[5].2   // Input Mayer Rod Operator Side Motor Overtemperature Warning
              p00_srv_mtr_os:I.DATA[5].3   // Input Mayer Rod Operator Side Reserved
              p00_srv_mtr_os:I.DATA[5].4   // Input Mayer Rod Operator Side Reserved
              p00_srv_mtr_os:I.DATA[5].5   // Input Mayer Rod Operator Side Position Velocity > Limit
              p00_srv_mtr_os:I.DATA[5].6   // Input Mayer Rod Operator Side Reserved
              p00_srv_mtr_os:I.DATA[5].7   // Input Mayer Rod Operator Side Reserved
              p00_srv_mtr_os:I.DATA[5].8   // Input Mayer Rod Operator Side Reserved
              p00_srv_mtr_os:I.DATA[5].9   // Input Mayer Rod Operator Side Undervoltage in DC bus
              p00_srv_mtr_os:I.DATA[5].10   // Input Mayer Rod Operator Side Reserved
              p00_srv_mtr_os:I.DATA[5].11   // Input Mayer Rod Operator Side Reserved
              p00_srv_mtr_os:I.DATA[5].12   // Input Mayer Rod Operator Side Reserved
              p00_srv_mtr_os:I.DATA[5].13   // Input Mayer Rod Operator Side Target Position Outside of position Limit Value
              p00_srv_mtr_os:I.DATA[5].14   // Input Mayer Rod Operator Side Reserved
              p00_srv_mtr_os:I.DATA[5].15   // Input Mayer Rod Operator Side Manufacturer - Specific Warning
              p00_srv_mtr_os:I.DATA[6]   // Input Mayer Rod Operator Side Diagnostic Message
              p00_srv_mtr_os:I   // Mayer Rod Operator Side
              p00_srv_mtr_os:O.DATA[0]   // Output Mayer Rod Operator Side VFD Control Word
              p00_srv_mtr_os:O.DATA[0].0   // Output Mayer Rod Operator Side Command Value Accept
              p00_srv_mtr_os:O.DATA[0].1   // Output Mayer Rod Operator Side OP/PM Mode Toggle
              p00_srv_mtr_os:O.DATA[0].2   // Output Mayer Rod Operator Side
              p00_srv_mtr_os:O.DATA[0].3   // Output Mayer Rod Operator Side
              p00_srv_mtr_os:O.DATA[0].4   // Output Mayer Rod Operator Side
              p00_srv_mtr_os:O.DATA[0].5   // Output Mayer Rod Operator Side Fault Reset
              p00_srv_mtr_os:O.DATA[0].6   // Output Mayer Rod Operator Side Jog Forward
              p00_srv_mtr_os:O.DATA[0].7   // Output Mayer Rod Operator Side Jog Reverse
              p00_srv_mtr_os:O.DATA[0].8   // Output Mayer Rod Operator Side Jog Enable
              p00_srv_mtr_os:O.DATA[0].9   // Output Mayer Rod Operator Side
              p00_srv_mtr_os:O.DATA[0].10   // Output Mayer Rod Operator Side
              p00_srv_mtr_os:O.DATA[0].11   // Output Mayer Rod Operator Side
              p00_srv_mtr_os:O.DATA[0].12   // Output Mayer Rod Operator Side
              p00_srv_mtr_os:O.DATA[0].13   // Output Mayer Rod Operator Side Drive Halt 0=Halt
              p00_srv_mtr_os:O.DATA[0].14   // Output Mayer Rod Operator Side Drive Enable
              p00_srv_mtr_os:O.DATA[0].15   // Output Mayer Rod Operator Side Drive On
              p00_srv_mtr_os:O.DATA[0].16   // Output Mayer Rod Operator Side Ready for Operation Bit 16 P-12 Bit 0
              p00_srv_mtr_os:O.DATA[0].17   // Output Mayer Rod Operator Side Ready for Operation Bit 17 P-12 Bit 1
              p00_srv_mtr_os:O.DATA[1]   // Output Mayer Rod Operator Side Velocity Command
              p00_srv_mtr_os:O.DATA[2]   // Output Mayer Rod Operator Side Position Command
              p00_srv_mtr_os:O.DATA[3]   // Output Mayer Rod Operator Side Jog Velocity Command
              p00_srv_mtr_os:O.DATA[4]   // Output Mayer Rod Operator Side Position Offset
              p00_srv_mtr_os:O   // Mayer Rod Operator Side
              p00_srv_mtr_os:C   // Mayer Rod Operator Side
         p00_srv_mtr_ds : ETHERNET-MODULE (Ethernet 10.0.1.16, rev 1.1, Output RPI 10 ms)
              p00_srv_mtr_ds:I.DATA[0]   // Input Mayer Rod Drive Side Status Word
              p00_srv_mtr_ds:I.DATA[0].0   // Input Mayer Rod Drive Side
              p00_srv_mtr_ds:I.DATA[0].1   // Input Mayer Rod Drive Side
              p00_srv_mtr_ds:I.DATA[0].2   // Input Mayer Rod Drive Side
              p00_srv_mtr_ds:I.DATA[0].3   // Input Mayer Rod Drive Side Stand Still
              p00_srv_mtr_ds:I.DATA[0].4   // Input Mayer Rod Drive Side Target Position Reached
              p00_srv_mtr_ds:I.DATA[0].5   // Input Mayer Rod Drive Side Command Change Bit
              p00_srv_mtr_ds:I.DATA[0].6   // Input Mayer Rod Drive Side Operating Mode Error
              p00_srv_mtr_ds:I.DATA[0].7   // Input Mayer Rod Drive Side Drive does not follow command value (e.g. when Drive Halt is active)
              p00_srv_mtr_ds:I.DATA[0].8   // Input Mayer Rod Drive Side Actual Operating Mode
              p00_srv_mtr_ds:I.DATA[0].9   // Input Mayer Rod Drive Side Actual Operating Mode
              p00_srv_mtr_ds:I.DATA[0].10   // Input Mayer Rod Drive Side
              p00_srv_mtr_ds:I.DATA[0].11   // Input Mayer Rod Drive Side Class 3 Diagnostic Message
              p00_srv_mtr_ds:I.DATA[0].12   // Input Mayer Rod Drive Side Class 2 Diagnostic Message
              p00_srv_mtr_ds:I.DATA[0].13   // Input Mayer Rod Drive Side Class 1 Diagnostic Message
              p00_srv_mtr_ds:I.DATA[0].14   // Input Mayer Rod Drive Side Ready for Operation Bit 14/15 00: Not Ready 01:(bb) 10: (Ab) 11: (AF)
              p00_srv_mtr_ds:I.DATA[0].15   // Input Mayer Rod Drive Side Ready for Operation Bit 14/15 00: Not Ready 01:(bb) 10: (Ab) 11: (AF)
              p00_srv_mtr_ds:I.DATA[1]   // Input Mayer Rod Drive Side Velocity Feedback
              p00_srv_mtr_ds:I.DATA[2]   // Input Mayer Rod Drive Side Position Feedback
              p00_srv_mtr_ds:I.DATA[3]   // Input Mayer Rod Drive Side Torque Feedback
              p00_srv_mtr_ds:I.DATA[4]   // Input Mayer Rod Drive Side Error Message
              p00_srv_mtr_ds:I.DATA[4].0   // Input Mayer Rod Drive Side Reserved
              p00_srv_mtr_ds:I.DATA[4].1   // Input Mayer Rod Drive Side Amplifier Overtemperature Shutdown
              p00_srv_mtr_ds:I.DATA[4].2   // Input Mayer Rod Operator Side Motot Overtemperature Shutdown
              p00_srv_mtr_ds:I.DATA[4].3   // Input Mayer Rod Drive Side Reserved
              p00_srv_mtr_ds:I.DATA[4].4   // Input Mayer Rod Drive Side Control Voltage Error
              p00_srv_mtr_ds:I.DATA[4].5   // Input Mayer Rod Drive Side Encoder Error
              p00_srv_mtr_ds:I.DATA[4].6   // Input Mayer Rod Drive Side Reserved
              p00_srv_mtr_ds:I.DATA[4].7   // Input Mayer Rod Drive Side Overcurrent Error
              p00_srv_mtr_ds:I.DATA[4].8   // Input Mayer Rod Drive Side Reserved
              p00_srv_mtr_ds:I.DATA[4].9   // Input Mayer Rod Drive Side Undervoltage Error
              p00_srv_mtr_ds:I.DATA[4].10   // Input Mayer Rod Drive Side Reserved
              p00_srv_mtr_ds:I.DATA[4].11   // Input Mayer Rod Drive Side Excessive Deviation
              p00_srv_mtr_ds:I.DATA[4].12   // Input Mayer Rod Drive Side Communication Error
              p00_srv_mtr_ds:I.DATA[4].13   // Input Mayer Rod Drive Side Position Limit Value Exceeded
              p00_srv_mtr_ds:I.DATA[4].14   // Input Mayer Rod Drive Side Reserved
              p00_srv_mtr_ds:I.DATA[4].15   // Input Mayer Rod Drive Side Manufacturer- Specific Error
              p00_srv_mtr_ds:I.DATA[5]   // Input Mayer Rod Drive Side Warning Message
              p00_srv_mtr_ds:I.DATA[5].0   // Input Mayer Rod Drive Side Overload Warning
              p00_srv_mtr_ds:I.DATA[5].1   // Input Mayer Rod Drive Side Amplifier Over Temp Warning
              p00_srv_mtr_ds:I.DATA[5].2   // Input Mayer Rod Drive Side Motor Over Temp Warning
              p00_srv_mtr_ds:I.DATA[5].3   // Input Mayer Rod Drive Side Reserved
              p00_srv_mtr_ds:I.DATA[5].4   // Input Mayer Rod Drive Side Reserved
              p00_srv_mtr_ds:I.DATA[5].5   // Input Mayer Rod Drive Side Positioning Vel > Limit
              p00_srv_mtr_ds:I.DATA[5].6   // Input Mayer Rod Drive Side Reserved
              p00_srv_mtr_ds:I.DATA[5].7   // Input Mayer Rod Drive Side Reserved
              p00_srv_mtr_ds:I.DATA[5].8   // Input Mayer Rod Drive Side Reserved
              p00_srv_mtr_ds:I.DATA[5].9   // Input Mayer Rod Drive Side Under Voltage in DC Bus
              p00_srv_mtr_ds:I.DATA[5].10   // Input Mayer Rod Drive Side Reserved
              p00_srv_mtr_ds:I.DATA[5].11   // Input Mayer Rod Drive Side Reserved
              p00_srv_mtr_ds:I.DATA[5].12   // Input Mayer Rod Drive Side Reserved
              p00_srv_mtr_ds:I.DATA[5].13   // Input Mayer Rod Drive Side Target Position outside of position limit values
              p00_srv_mtr_ds:I.DATA[5].14   // Input Mayer Rod Drive Side Reserved
              p00_srv_mtr_ds:I.DATA[5].15   // Input Mayer Rod Drive Side Manufacturer Specific Warning
              p00_srv_mtr_ds:I.DATA[6]   // Input Mayer Rod Drive Side Diagnostic Message
              p00_srv_mtr_ds:I   // Mayer Rod Drive Side
              p00_srv_mtr_ds:O.DATA[0]   // Output Mayer Rod Drive Side Control Word
              p00_srv_mtr_ds:O.DATA[0].0   // Output Mayer Rod Drive Side Command Value Accept
              p00_srv_mtr_ds:O.DATA[0].1   // Output Mayer Rod Drive Side
              p00_srv_mtr_ds:O.DATA[0].2   // Output Mayer Rod Drive Side
              p00_srv_mtr_ds:O.DATA[0].3   // Output Mayer Rod Drive Side
              p00_srv_mtr_ds:O.DATA[0].4   // Output Mayer Rod Drive Side
              p00_srv_mtr_ds:O.DATA[0].5   // Output Mayer Rod Drive Side Fault Reset
              p00_srv_mtr_ds:O.DATA[0].6   // Output Mayer Rod Drive Side Jog Forward
              p00_srv_mtr_ds:O.DATA[0].7   // Output Mayer Rod Drive Side Jog Reverse
              p00_srv_mtr_ds:O.DATA[0].8   // Output Mayer Rod Drive Side Jog Enable
              p00_srv_mtr_ds:O.DATA[0].9   // Output Mayer Rod Drive Side
              p00_srv_mtr_ds:O.DATA[0].10   // Output Mayer Rod Drive Side
              p00_srv_mtr_ds:O.DATA[0].11   // Output Mayer Rod Drive Side
              p00_srv_mtr_ds:O.DATA[0].12   // Output Mayer Rod Drive Side
              p00_srv_mtr_ds:O.DATA[0].13   // Output Mayer Rod Drive Side Drive Halt 0=Halt
              p00_srv_mtr_ds:O.DATA[0].14   // Output Mayer Rod Drive Side Drive Enable
              p00_srv_mtr_ds:O.DATA[0].15   // Output Mayer Rod Drive Side
              p00_srv_mtr_ds:O.DATA[0].16   // Output Mayer Rod Drive Sied Ready for Operation Bit 16 P-12 Bit 0
              p00_srv_mtr_ds:O.DATA[0].17   // Output Mayer Rod Drive Sied Ready for Operation Bit 17 P-12 Bit 1
              p00_srv_mtr_ds:O.DATA[1]   // Output Mayer Rod Drive Side Velocity Command
              p00_srv_mtr_ds:O.DATA[2]   // Output Mayer Rod Drive Side Position Command
              p00_srv_mtr_ds:O.DATA[3]   // Output Mayer Rod Drive Side Jog Velocity Command
              p00_srv_mtr_ds:O.DATA[4]   // Output Mayer Rod Drive Side Position Offset
              p00_srv_mtr_ds:O   // Mayer Rod Drive Side Servo
              p00_srv_mtr_ds:C   // Mayer Rod Drive Side
         p00_vfd_ts2 : ETHERNET-MODULE (Ethernet 10.0.1.17, rev 1.1, Output RPI 10 ms)
              p00_vfd_ts2:C   // Tension Stand 2 VFD
         p00_vfd_slitter : ETHERNET-MODULE (Ethernet 10.0.1.18, rev 1.1, Output RPI 10 ms)
              p00_vfd_slitter:I.DATA[0]   // Input Slitter VFD Status Word
              p00_vfd_slitter:I.DATA[0].0   // Input Slitter VFD Faulted
              p00_vfd_slitter:I.DATA[0].1   // Input Slitter VFD Warning
              p00_vfd_slitter:I.DATA[0].2   // Input Slitter VFD Running Forward
              p00_vfd_slitter:I.DATA[0].3   // Input Slitter VFD Running Reverse
              p00_vfd_slitter:I.DATA[0].4   // Input Slitter VFD Ready
              p00_vfd_slitter:I.DATA[0].5   // Input Slitter VFD Control from Net
              p00_vfd_slitter:I.DATA[0].6   // Input Slitter VFD Reference from Net
              p00_vfd_slitter:I.DATA[0].7   // Input Slitter VFD At Reference
              p00_vfd_slitter:I.DATA[1]   // Input Slitter VFD Speed
              p00_vfd_slitter:I.DATA[2]   // Input Slitter VFD Amps
              p00_vfd_slitter:I.DATA[3]   // Input Slitter VFD Max Hertz
              p00_vfd_slitter:I.DATA[4]   // Input Slitter VFD Motor Nameplate Hertz
              p00_vfd_slitter:I.DATA[5]   // Input Slitter VFD Motor Nameplate RPM
              p00_vfd_slitter:I   // Slitter VFD
              p00_vfd_slitter:O.DATA[0]   // Output Slitter VFD Control Word
              p00_vfd_slitter:O.DATA[0].0   // Output Slitter VFD Run Forward
              p00_vfd_slitter:O.DATA[0].1   // Output Slitter VFD Run Reverse
              p00_vfd_slitter:O.DATA[0].2   // Output Slitter VFD Fault Reset
              p00_vfd_slitter:O.DATA[0].5   // Output Slitter VFD Net Control
              p00_vfd_slitter:O.DATA[0].6   // Output Slitter VFD Net Reference
              p00_vfd_slitter:O.DATA[1]   // Output Slitter VFD Speed Command
              p00_vfd_slitter:O   // Slitter VFD
              p00_vfd_slitter:C   // Slitter VFD
         p00_vfd_wdr_turret : ETHERNET-MODULE (Ethernet 10.0.1.19, rev 1.1, Output RPI 10 ms)
              p00_vfd_wdr_turret:I.DATA[0]   // Input Winder Turret VFD Status Word
              p00_vfd_wdr_turret:I.DATA[0].0   // Input Winder Turret VFD Faulted
              p00_vfd_wdr_turret:I.DATA[0].1   // Input Winder Turret VFD Warning
              p00_vfd_wdr_turret:I.DATA[0].2   // Input Winder Turret VFD Running Forward
              p00_vfd_wdr_turret:I.DATA[0].3   // Input Winder Turret VFD Running Reverse
              p00_vfd_wdr_turret:I.DATA[0].4   // Input Winder Turret VFD Ready
              p00_vfd_wdr_turret:I.DATA[0].5   // Input Winder Turret VFD Control from Net
              p00_vfd_wdr_turret:I.DATA[0].6   // Input Winder Turret VFD Reference from Net
              p00_vfd_wdr_turret:I.DATA[0].7   // Input Winder Turret VFD At Reference
              p00_vfd_wdr_turret:I.DATA[1]   // Input Winder Turret VFD Speed
              p00_vfd_wdr_turret:I.DATA[2]   // Input Winder Turret VFD Amps
              p00_vfd_wdr_turret:I.DATA[3]   // Input Winder Turret VFD Max Hertz
              p00_vfd_wdr_turret:I.DATA[4]   // Input Winder Turret VFD Motor Nameplate Hertz
              p00_vfd_wdr_turret:I.DATA[5]   // Input Winder Turret VFD Motor Nameplate RPM
              p00_vfd_wdr_turret:I   // Winder Turret VFD
              p00_vfd_wdr_turret:O.DATA[0]   // Output Winder Turret VFD Control Word
              p00_vfd_wdr_turret:O.DATA[0].0   // Output Winder Turret VFD Run Forward
              p00_vfd_wdr_turret:O.DATA[0].1   // Output Winder Turret VFD Run Reverse
              p00_vfd_wdr_turret:O.DATA[0].2   // Output Winder Turret VFD Fault Reset
              p00_vfd_wdr_turret:O.DATA[0].5   // Output Winder Turret VFD Net Control
              p00_vfd_wdr_turret:O.DATA[0].6   // Output Winder Turret VFD Net Reference
              p00_vfd_wdr_turret:O.DATA[1]   // Output Winder Turret VFD Speed Command
              p00_vfd_wdr_turret:O   // Winder Turret VFD
              p00_vfd_wdr_turret:C   // Winder Turret VFD
         p00_vfd_wda : ETHERNET-MODULE (Ethernet 10.0.1.20, rev 1.1, Output RPI 10 ms)
              p00_vfd_wda:I.DATA[0]   // Output Tension Stand 2 VFD Control Word
              p00_vfd_wda:I.DATA[0].0   // Output Tension Stand 2 VFD Run Forward
              p00_vfd_wda:I.DATA[0].1   // Output Tension Stand 2 VFD Run Reverse
              p00_vfd_wda:I.DATA[0].2   // Output Tension Stand 2 VFD Fault Reset
              p00_vfd_wda:I.DATA[0].5   // Output Tension Stand 2 VFD Net Control
              p00_vfd_wda:I.DATA[0].6   // Output Tension Stand 2 VFD Net Reference
              p00_vfd_wda:I.DATA[1]   // Output Tension Stand 2 VFD Speed Command
              p00_vfd_wda:I   // Tension Stand 2 VFD
              p00_vfd_wda:C   // Winder A VFD
         p00_vfd_sprng : ETHERNET-MODULE (Ethernet 10.0.1.22, rev 1.1, Output RPI 10 ms)
         T000_ENC_Winder : 843E-MIPxxBAx (Ethernet 10.0.1.23, rev 1.1, StandardDataDriven RPI 25 ms)   // Winder Turret
      p00_ai_01 : 1756-IF16 (ICP 3, rev 1.1, Input RPI 100 ms)
           Local:3:I.CH0DATA   // Analog Input Tension Stand 1 Load Cell
           Local:3:I.CH1DATA   // Analog Input Splice Press Load Cell
           Local:3:I.CH2DATA   // Analog Input Winder Stand Load Cell
           Local:3:I.CH3DATA   // Analog Input Spare
           Local:3:I.CH4DATA   // Analog Input Letoff A Yardage
           Local:3:I.CH5DATA   // Analog Input Letoff B Yardage
           Local:3:I.CH6DATA   // Analog Input Winder A Yardage
           Local:3:I.CH7DATA   // Analog Input Winder B Yardage
END_MODULES
